FUNCTION_BLOCK HighestRequestProducer
  (* Standard: 61499-2 *)
  (* Version 0.1, 2014-00-16, Canto-Air, CANTO-AIR-PC *)
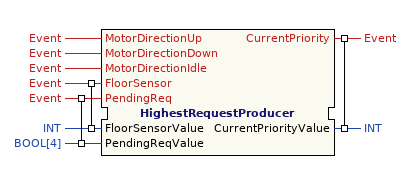
  EVENT_INPUT
    MotorDirectionUp;
    MotorDirectionDown;
    MotorDirectionIdle;
    FloorSensor WITH FloorSensorValue;
    PendingReq WITH PendingReqValue;
  END_EVENT
  EVENT_OUTPUT
    CurrentPriority WITH CurrentPriorityValue;
  END_EVENT
  VAR_INPUT
    FloorSensorValue : INT;
    PendingReqValue : ARRAY [0..3] OF BOOL;
  END_VAR
  VAR_OUTPUT
    CurrentPriorityValue : INT;
  END_VAR
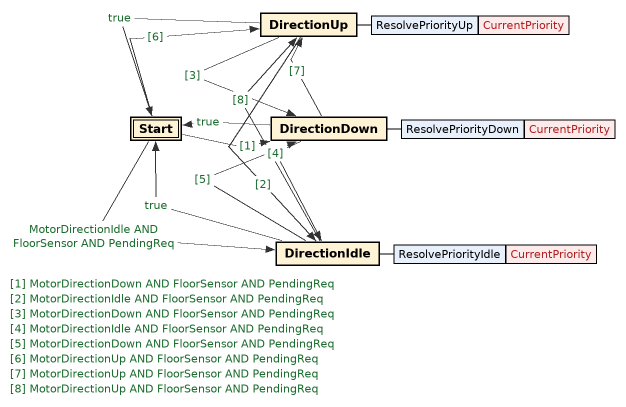
  EC_STATES
    Start;
    DirectionUp : ResolvePriorityUp -> CurrentPriority;
    DirectionDown : ResolvePriorityDown -> CurrentPriority;
    DirectionIdle : ResolvePriorityIdle -> CurrentPriority;
  END_STATES
  EC_TRANSITIONS
    Start TO DirectionUp := MotorDirectionUp AND FloorSensor AND PendingReq;
    Start TO DirectionDown := MotorDirectionDown AND FloorSensor AND PendingReq;
    Start TO DirectionIdle := MotorDirectionIdle AND FloorSensor AND PendingReq;
    DirectionUp TO DirectionIdle := MotorDirectionIdle AND FloorSensor AND PendingReq;
    DirectionUp TO DirectionDown := MotorDirectionDown AND FloorSensor AND PendingReq;
    DirectionUp TO Start := true;
    DirectionDown TO DirectionUp := MotorDirectionUp AND FloorSensor AND PendingReq;
    DirectionDown TO DirectionIdle := MotorDirectionIdle AND FloorSensor AND PendingReq;
    DirectionDown TO Start := true;
    DirectionIdle TO DirectionUp := MotorDirectionUp AND FloorSensor AND PendingReq;
    DirectionIdle TO DirectionDown := MotorDirectionDown AND FloorSensor AND PendingReq;
    DirectionIdle TO Start := true;
  END_TRANSITIONS
  ALGORITHM ResolvePriorityUp IN C:
int bitmask;
int PendingReq = 0;
int i = 0;
me->CurrentPriorityValue = -1;
for (i = 0; i < 4; ++i) {
    PendingReq |= me->PendingReqValue[i] << i;
}
printf("Pending Request, direction, current: %d 1 %d\n", PendingReq, me->FloorSensorValue);
// initial condition => priority hasn't been changed
me->CurrentPriorityValue = -1;
bitmask = 0x01;
for (i = 0 ; i < 4; ++i) {
    if (i > me->FloorSensorValue && (PendingReq & bitmask)) {
        me->CurrentPriorityValue = i;
        printf("Up Priority = %d\n", me->CurrentPriorityValue );
        break;
    }
    bitmask = bitmask << 1;
}
  END_ALGORITHM
  ALGORITHM ResolvePriorityDown IN C:
int bitmask;
int PendingReq = 0;
int i = 0;
me->CurrentPriorityValue = -1;
for (i = 0; i < 4; ++i) {
    PendingReq |= me->PendingReqValue[i] << i;
}
printf("Pending Request, direction, current: %d 2 %d\n", PendingReq, me->FloorSensorValue);
bitmask = 0x08;
for (i = 4 - 1; i > -1; --i) {
    if (i < me->FloorSensorValue && (PendingReq & bitmask)) {
        me->CurrentPriorityValue  = i;
        printf("Down Priority = %d\n", me->CurrentPriorityValue );
        break;
    }
    bitmask = bitmask >> 1;
}
  END_ALGORITHM
  ALGORITHM ResolvePriorityIdle IN C:
int bitmask;
int PendingReq = 0;
int i = 0;
me->CurrentPriorityValue = -1;
for (i = 0; i < 4; ++i) {
    PendingReq |= me->PendingReqValue[i] << i;
}
printf("Pending Request, direction, current: %d 3 %d\n", PendingReq, me->FloorSensorValue);
printf("Current %d \n", me->FloorSensorValue);
if (me->FloorSensorValue == 0) {
    printf("Idle case when on bottom floor\n");
    bitmask = 0x01;
    for (i = 0; i < 4; ++i) {
        if (i > me->FloorSensorValue && (PendingReq & bitmask)) {
            me->CurrentPriorityValue = i;
            printf("Init Up Priority = %d\n", me->CurrentPriorityValue);
            break;
        }
        bitmask = bitmask << 1;
    }
} else if (me->FloorSensorValue == 4 - 1) {
    printf("Idle case when on top floor\n");
    bitmask = 0x08;
    for (i = 4 - 1; i > -1; --i) {
        if (i < me->FloorSensorValue && (PendingReq & bitmask)) {
            me->CurrentPriorityValue = i;
            printf("Init Down Priority= %d\n", me->CurrentPriorityValue);
            break;
        }
        bitmask = bitmask >> 1;
    }
} else {
    //if lift is somewhere in the middle it will go down if
    //there is any requests below the current floor
    printf("Idle case when on some middle floor\n");
    bitmask = 0x01;
    for (i = 0; i < 4; ++i) {
        if (i > me->FloorSensorValue && (PendingReq & bitmask)) {
            me->CurrentPriorityValue = i;
            printf("Middle Up Priority = %d\n", me->CurrentPriorityValue);
            break;
        }
        bitmask = bitmask << 1;
    }
    // if there are no up requests > current
    if (me->CurrentPriorityValue == -1) {
        bitmask = 0x08;
        for(i = 4- 1; i > -1; --i) {
            if (i < me->FloorSensorValue && (PendingReq & bitmask)) {
                me->CurrentPriorityValue = i;
                printf("Middle Down Priority = %d\n", me->CurrentPriorityValue);
                break;
            }
            bitmask = bitmask >> 1;
        }
    }
}
  END_ALGORITHM
END_FUNCTION_BLOCK
